PROGRAM POU_Test
VAR
	readBuff:ARRAY [1..10] OF ST_DataFmtBase;
	fbFileReadWrite:FB_IOFileReadWrite;
END_VAR

fbFileReadWrite(
	readBuff:= readBuff, 
	sFileName:= 'E:\FilePath\file.csv', 
	bRead:= , 
	sTxtHead:= 'GROUP,NUM,ENG,CHN,NO USE', 
	bBusy=> , 
	bDone=> , 
	bError=> , 
	nErrid=> );

END_PROGRAM

(* stored: Version 1.1.0.1, ProductVersion 3.1.4024.4
   POU POU_Test: Id {0b577caa-b73d-4a1d-80e9-1a9aceb2b453}, SpecialFunc None *)
